(* CODESYS project festo_cmmt_as.library
   Title: FESTO CMMT_AS Drive Control
   Version: 1.0
   Placeholder: FESTO CMMT_AS Drive Control
   Company: Sensata Mech Sofia

Project tree, tasks and I/O mapping:
  libraries: Festo_PtP_Base, * (Festo); Festo_PtP_CiA402, * (Festo); Festo_PtP_CiA402_ETC, * (Festo); Festo_PtP_CiA402_ETC_CMMT_AS, * (Festo); Festo_PtP_Virtual, * (Festo); Tc2_Standard, * (Beckhoff Automation GmbH); Tc2_System, * (Beckhoff Automation GmbH); Tc3_Module, * (Beckhoff Automation GmbH)
  DUTs/
    data type driveStates
  GVLs/
  POUs/
    function block FB_FESTO_CMMT_AS [ST]
  VISUs/
*)

// DUTs/driveStates
{attribute 'qualified_only'}
{attribute 'strict'}
TYPE driveStates :
(
	stStartUp 			:= 0,
	stStandStill,
	stHoming,
	stDisable,
	stErrorStop,
	stStopping, 
	stMotion
	
);
END_TYPE

// POUs/FB_FESTO_CMMT_AS
FUNCTION_BLOCK FB_FESTO_CMMT_AS

VAR_INPUT
	
	axis 					:  REFERENCE TO  AXIS_REF_CiA402_ETC_CMMT_AS;
	PowerUp                 :  BOOL;
	Home                    :  BOOL;
	StartMove               :  BOOL;
	Reset                   :  BOOL;
	Position                :  REAL;
	Velocity                :  REAL;
	Acceleration            :  REAL;
	IsAbsolute              :  BOOL;
	
END_VAR

VAR_OUTPUT
	
	Enabled                 :  BOOL;
	Error                   :  BOOL;
	ErrorID                 :  UDINT;
	TargetReached           :  BOOL;
	HomeDone                :  BOOL;
	Moving                  :  BOOL;
	CurrentPosition         :  REAL;
	OperationMode           :  UDINT;

END_VAR

VAR

	activeState              : driveStates; 
	fbError                  : MC_ReadAxisError_Festo;
	fbCurrentPos             : MC_ReadActualPosition_Festo;
	fbPower                  : MC_Power_Festo;
	fbReset                  : MC_Reset_Festo;
	fbHome                   : MC_Home_Festo;
	fbMove                   : MC_MoveAbsolute_Festo;

	doDisMove                 : BOOL;
	doHoming				  : BOOL;
	
END_VAR


axis();

fbError(Axis:=axis, Enable:=TRUE);

IF fbError.Valid AND fbError.AxisErrorID <> 0 THEN
	Error       := TRUE;
	ErrorID     := fbError.ErrorID;
	activeState := driveStates.stErrorStop;
END_IF

fbMove(Axis:=axis,  Execute:=doDisMove, Position:= Position, Velocity:=Velocity, Acceleration:=Acceleration, Deceleration:=Acceleration);
fbHome(Axis:=axis,  Execute:=doHoming,  Position:=0, HomingMethod:=0);
fbReset(Axis:=axis, Execute:=Reset);
fbPower(Axis:=axis, Enable:=PowerUp);

IF NOT fbPower.Status AND fbError.Valid AND fbError.AxisErrorID = 0 THEN
	activeState := driveStates.stDisable;
END_IF

fbCurrentPos(Axis:=axis, Enable:=TRUE);

IF fbCurrentPos.Valid THEN
	CurrentPosition := fbCurrentPos.Position;
END_IF

IF fbMove.Active OR fbHome.Active THEN
	Moving := TRUE;
ELSE
	Moving := FALSE;
END_IF

IF IsAbsolute THEN
	OperationMode := 0;
	IF NOT fbHome.Active THEN
		HomeDone := TRUE;
	END_IF
ELSE
	OperationMode := 1;
END_IF

CASE activeState OF
	
	driveStates.stErrorStop:
		Moving  := FALSE;
		IF NOT fbPower.Status AND fbReset.Done THEN
			activeState := driveStates.stDisable;
		ELSIF fbPower.Status AND fbPower.Enable AND fbPower.valid AND fbReset.Done THEN
			activeState := driveStates.stStandStill;
		END_IF
	
	driveStates.stDisable:
		Error   := FALSE;
		ErrorID := 0;
		Enabled := FALSE;
		IF fbPower.valid AND fbPower.Status AND fbPower.Enable THEN
			activeState := driveStates.stStandStill;
		END_IF
	
	driveStates.stStandStill:
		Error     := FALSE;
		ErrorID   := 0;
		doDisMove := StartMove;
		doHoming  := Home;
		Enabled   := TRUE;
		IF fbHome.Active THEN
			HomeDone    := FALSE;
			activeState := driveStates.stHoming;
		END_IF
		IF fbMove.Active THEN
			TargetReached := FALSE;
			activeState := driveStates.stMotion;		
		END_IF
		
	driveStates.stMotion:
		IF fbMove.Done THEN
			TargetReached := TRUE;
			activeState   := driveStates.stStandStill;
		END_IF
		
	driveStates.stHoming:
		IF fbHome.Done THEN
			HomeDone    := TRUE;
			activeState := driveStates.stStandStill;
		END_IF
		
END_CASE

END_FUNCTION_BLOCK
